{attribute 'qualified_only'}
VAR_GLOBAL
	Vessel : ARRAY [1..2] OF TYP_VESSEL_HW;
	Buttons : TYP_BUTTONS_HW_IN;
	
END_VAR

(* stored: Version 1.1.0.1, ProductVersion 3.1.4024.12
   GVL gOpc: Id {75962204-cf7b-4a17-b9d9-6bdb8cdb3d0e} *)
